// TIA Portal V20 export
// export: Created 2025-12-01T14:56:10.3661262Z, ExportSetting None, DisplayName Totally Integrated Automation Portal, DisplayVersion V20 Update 3, DisplayName TIA Portal Openness, DisplayVersion V20 Update 3, DisplayName TIA Portal Version Control Interface, DisplayVersion V20 Update 3, DisplayName STEP 7 Professional, DisplayVersion V20 Update 3, DisplayName STEP 7 Safety, DisplayVersion V20 Update 2, DisplayName WinCC Basic/Comfort/Advanced, DisplayVersion V20 Update 3, DisplayName WinCC Professional, DisplayVersion V20 Update 3, DisplayName WinCC Unified, DisplayVersion V20 Update 3
TYPE "LPNDR_typePortLinkState"
   STRUCT
      portName : String[14];
      portLinkState : Byte;   // 1=up, 2=Down, 3=testing, 4=unknown, 5=dormant, 6= notPresent, 7=LowerLayerDown
      portPortState : Byte;
   END_STRUCT;
END_TYPE
